// Mitsubishi GX Works2 project: DZRN_DDRVA_automove_p1   PLC: FX3U/FX3UC

PROGRAM MAIN
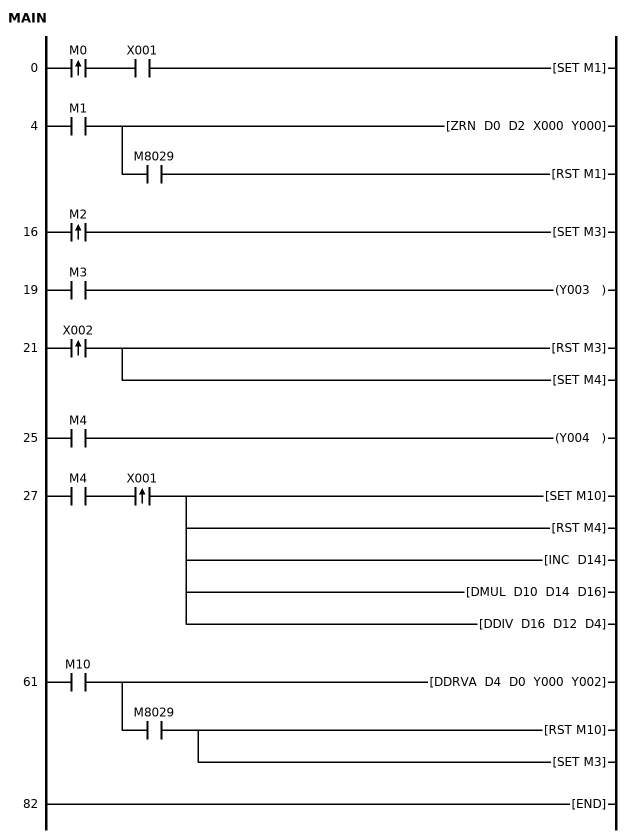
0     LDP     M0
      AND     X001
      SET     M1
4     LD      M1
      ZRN     D0 D2 X000 Y000
      AND     M8029
      RST     M1
16    LDP     M2
      SET     M3
19    LD      M3
      OUT     Y003
21    LDP     X002
      RST     M3
      SET     M4
25    LD      M4
      OUT     Y004
27    LD      M4
      ANDP    X001
      SET     M10
      RST     M4
      INC     D14
      DMUL    D10 D14 D16
      DDIV    D16 D12 D4
61    LD      M10
      DDRVA   D4 D0 Y000 Y002
      AND     M8029
      RST     M10
      SET     M3
82    END
END_PROGRAM
